{attribute 'GeneratedUsingTerminal: EK1100-0000-0018'}
{attribute addProperty BoxType "EK1100-0000-0018"}
{attribute addProperty Id "A_0016_BK1250_0000_0017A_0016_BK1250_0000_0017_C46DBFF00"}
{attribute addProperty CRC "1905245092"}
{attribute addProperty Size "0"}
{attribute addProperty Name "Term 19 (EK1100)"}
TYPE Term_19_EK1100_718FBBA4 EXTENDS EK1100_1FC0878B :
STRUCT
	{attribute addProperty Name "A_0016(BK1250-0000-0017)"}
	{attribute addProperty PreviousPort "Term 19 (EK1100) : B"}
	A_0016_BK1250_0000_0017 : A_0016_BK1250_0000_0017_C46DBFF0;
END_STRUCT
END_TYPE

(* stored: Version 1.2.0.0, ProductVersion 3.1.4024.11
   DUT Term_19_EK1100_718FBBA4: Id {a7618198-49d3-438f-b3fc-8d35961df07f} *)
